TYPE ST_HeatPumpDefaultParameters :
STRUCT
	aSetPointLimitsTemperature : ARRAY[1..2] OF REAL := [10,100]; //setpoint limits for tsupply temperature
END_STRUCT
END_TYPE

(* stored: Version 1.1.0.1, ProductVersion 3.1.4024.10
   DUT ST_HeatPumpDefaultParameters: Id {9f6c8311-4370-4841-8890-344d838cbcd7} *)
